ABB RobotStudio station: RoboEdgeMapping.rsstnx

Station RoboEdgeMapping (saved by RobotStudio 23.2.10478.1)
Controller IRB120_3_58
  mechanical unit ROB_1: IRB120T_3_58__01, 6 joints, base frame (0, 0, 0) mm
Layout (positions relative to the parent item):
  - IRB120T_3_58__01 [mechanism, from %ABB.RobotStudio.Models.IRB120%\IRB120T_3_58_G_01.rslib] at (0, 0, 0) mm; joint values [0.1026, 0.6018, -0.3453, -0.1035, 0.6562, 0.1631] (rad or m)
  - MyTool [mechanism, from Training Objects\myTool.rslib] at (395.28, 47.39, 446.93) mm, rotated rx 180 ry 38 rz 180 deg
  - Part_1 [part]
  - Part_2 [part] at (150, -20, 0) mm, size 138.5 x 87.5 x 246.4 mm
Attachment: MyTool is attached to IRB120T_3_58__01 / Link6
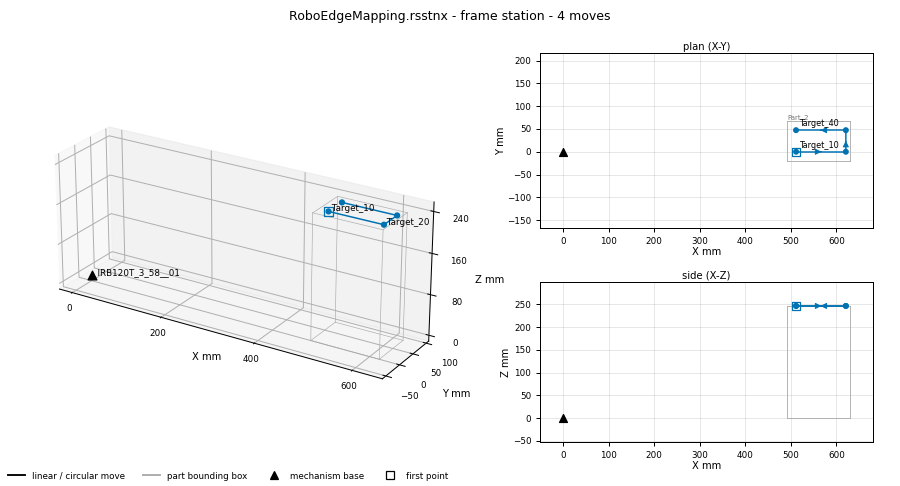
[picture p0: tool path of RoboEdgeMapping.rsstnx in frame station, 4 of 4 moves have a stored position in this frame; points joined in program order, loops and branches not executed]
Targets, tools, work objects and paths stored in the station, written as RAPID:
! task T_ROB1
MODULE CalibData
  PERS tooldata MyTool:=[TRUE,[[31.792631019,0,229.638935148],[0.945518576,0,0.325568154,0]],[1,[0,0,1],[1,0,0,0],0,0,0]];
  TASK PERS wobjdata Workobject_Box:=[FALSE,TRUE,"",[[511.6,0,246.399],[1,0,0,0]],[[0,0,0],[1,0,0,0]]];
ENDMODULE

! task T_ROB1
MODULE Module1
  CONST robtarget Target_10:=[[0.091,0,0.003],[0,0,1,0],[0,0,0,0],[9E+09,9E+09,9E+09,9E+09,9E+09,9E+09]];
  CONST robtarget Target_20:=[[109.303,0,0.003],[0,0,1,0],[0,0,-1,0],[9E+09,9E+09,9E+09,9E+09,9E+09,9E+09]];
  CONST robtarget Target_30:=[[109.35,47.385,0.003],[0,0,1,0],[0,-1,0,0],[9E+09,9E+09,9E+09,9E+09,9E+09,9E+09]];
  CONST robtarget Target_40:=[[0.006,47.385,0.003],[0,0,1,0],[0,-1,0,0],[9E+09,9E+09,9E+09,9E+09,9E+09,9E+09]];
  PROC Path_10()
    MoveL Target_10,v500,fine,MyTool\WObj:=Workobject_Box;
    MoveL Target_20,v500,fine,MyTool\WObj:=Workobject_Box;
    MoveL Target_30,v500,fine,MyTool\WObj:=Workobject_Box;
    MoveL Target_40,v500,fine,MyTool\WObj:=Workobject_Box;
  ENDPROC
  PROC main()
    Path_10;
  ENDPROC
ENDMODULE

